(* PLC project Generated.project, CODESYS CODESYS V3.5 SP19 Patch 1 *)
(* stored: creationDateTime 2026-08-18T01:34:50.927930, modificationDateTime 2026-08-18T01:34:50.927930 *)

(* ═══════════════════════════════════════════════════════════════ ST_DredgingAssistCfg — Réglages persistants assistants prélèvement 📄 Doc : DOC/AF/AF_Partie-04_Mode_SemiAuto_Sequenceur_v2.1.md §3ter ═══════════════════════════════════════════════════════════════ *)
TYPE ST_DredgingAssistCfg : STRUCT
  DiveStartMin_M : REAL := 1;  (* Position mini M1/M2 avant plongée *)
  ImmersionUpper_M : REAL := 0.5;  (* Borne haute fenêtre front immersion *)
  ImmersionLower_M : REAL := -0.5;  (* Borne basse fenêtre front immersion *)
  ExtractionControlDistance_M : REAL := 2;  (* Remontée palier 1 avant accélération *)
  TglEnableDiveSearch : BOOL := FALSE;  (* Mode assistance plongée mémorisé *)
  TglEnableExtractionSequence : BOOL := FALSE;  (* Mode assistance extraction mémorisé *)
  TglEnableDumpAtTremie : BOOL := FALSE;  (* Mode assistance vidage trémie mémorisé *)
  Initialized : BOOL := FALSE;  (* Pont persistance/IHM initialisé *)
END_STRUCT;
END_TYPE

(* ======================================================================= 💾 FB_CfgPersistBridge_DredgingAssistCfg — Pont persistance prélèvement ─────────────────────────────────────────────────────────────── 🎯 Rôle : Restauration et synchronisation bidirectionnelle IHM / Persist 💾 Persistance : Transfert GVL_PERSISTENT <-> GVL_IHM sur Initialized 📄 Doc métier : DOC/AF/AF_Partie-03_Contrats_Composants_v2.1.md §3 ======================================================================= *)
FUNCTION_BLOCK FB_CfgPersistBridge_DredgingAssistCfg
  VAR_OUTPUT
    JustRestored : BOOL;  (* === ETATS RESTAURATION === <-- [STAT] Vrai sur le cycle de restauration initiale *)
  END_VAR
  VAR_IN_OUT
    Hmi : ST_DredgingAssistCfg;  (* === BUS CONFIGURATION ET PERSISTANCE === <-> [BUS] Structure de configuration IHM *)
    Persist : ST_DredgingAssistCfg;  (* <-> [BUS] Structure de configuration persistante *)
  END_VAR

            

JustRestored := FALSE;
IF NOT Hmi.Initialized THEN
    Hmi := Persist;
    Hmi.Initialized := TRUE;
    JustRestored := TRUE;
ELSE
    Persist := Hmi;
END_IF;

          
END_FUNCTION_BLOCK
